TYPE (* IEC 61131-3-2.3.3.2 *)
  (* Standard: 61131-3 *)
  (* Version 0.1, 2000-05-16, JHC, Rockwell Automation, File type changed to ".dtp" *)
  (* Version 0.0, 2000-04-19, JHC, Rockwell Automation *)
  (* Compiler header: package fb.rt.ita; *)
  (* ASN.1 tag PRIVATE 15 *)
  ANALOG_16_INPUT_DATAI : ARRAY [0..15] OF ANALOG_DATA := [8(-4095),8(4095)];
END_TYPE
